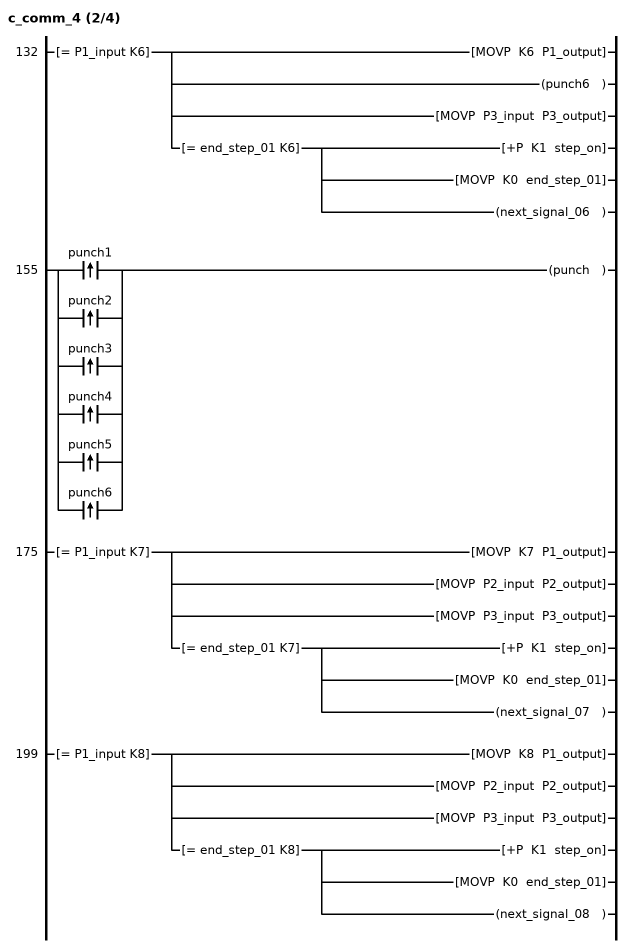
[picture p48: ladder of c_comm_4, rungs at steps 132 to 199]
132   LD=     P1_input K6
      MOVP    K6 P1_output
      OUT     punch6
      MOVP    P3_input P3_output
      AND=    end_step_01 K6
      +P      K1 step_on
      MOVP    K0 end_step_01
      OUT     next_signal_06
155   LDP     punch1
      ORP     punch2
      ORP     punch3
      ORP     punch4
      ORP     punch5
      ORP     punch6
      OUT     punch
175   LD=     P1_input K7
      MOVP    K7 P1_output
      MOVP    P2_input P2_output
      MOVP    P3_input P3_output
      AND=    end_step_01 K7
      +P      K1 step_on
      MOVP    K0 end_step_01
      OUT     next_signal_07
199   LD=     P1_input K8
      MOVP    K8 P1_output
      MOVP    P2_input P2_output
      MOVP    P3_input P3_output
      AND=    end_step_01 K8
      +P      K1 step_on
      MOVP    K0 end_step_01
      OUT     next_signal_08
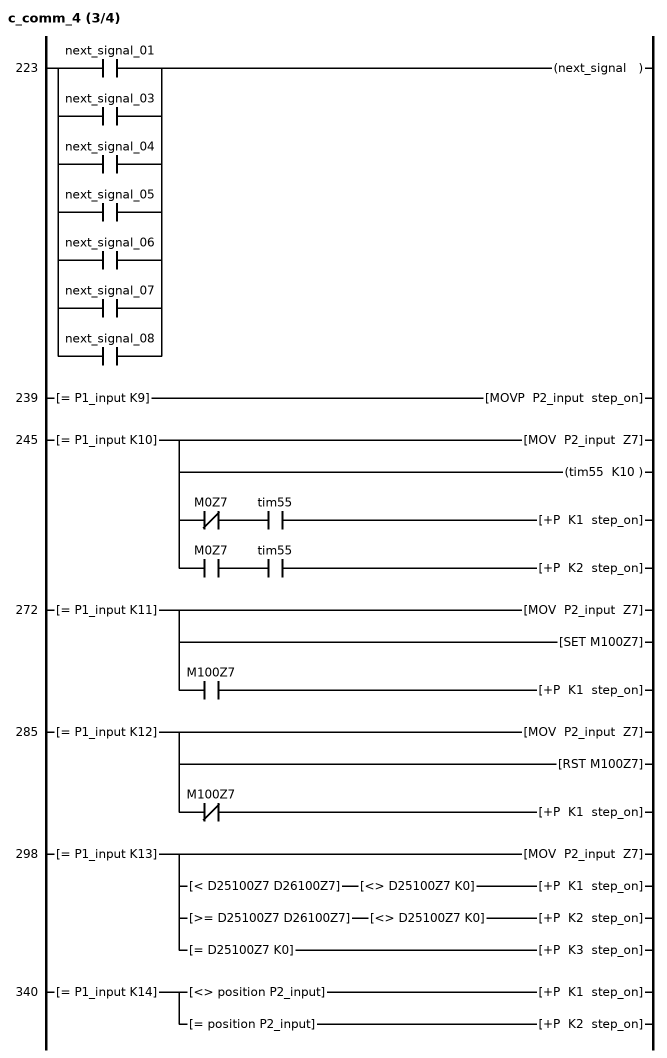
223   LD      next_signal_01
      OR      next_signal_03
      OR      next_signal_04
      OR      next_signal_05
      OR      next_signal_06
      OR      next_signal_07
      OR      next_signal_08
      OUT     next_signal
239   LD=     P1_input K9
      MOVP    P2_input step_on
245   LD=     P1_input K10
      MOV     P2_input Z7
      OUT     tim55 K10
      MPS
      ANI     M0Z7
      AND     tim55
      +P      K1 step_on
      MPP
      AND     M0Z7
      AND     tim55
      +P      K2 step_on
272   LD=     P1_input K11
      MOV     P2_input Z7
      SET     M100Z7
      AND     M100Z7
      +P      K1 step_on
285   LD=     P1_input K12
      MOV     P2_input Z7
      RST     M100Z7
      ANI     M100Z7
      +P      K1 step_on
298   LD=     P1_input K13
      MOV     P2_input Z7
      MPS
      AND<    D25100Z7 D26100Z7
      AND<>   D25100Z7 K0
      +P      K1 step_on
      MRD
      AND>=   D25100Z7 D26100Z7
      AND<>   D25100Z7 K0
      +P      K2 step_on
      MPP
      AND=    D25100Z7 K0
      +P      K3 step_on
340   LD=     P1_input K14
      MPS
      AND<>   position P2_input
      +P      K1 step_on
      MPP
      AND=    position P2_input
      +P      K2 step_on
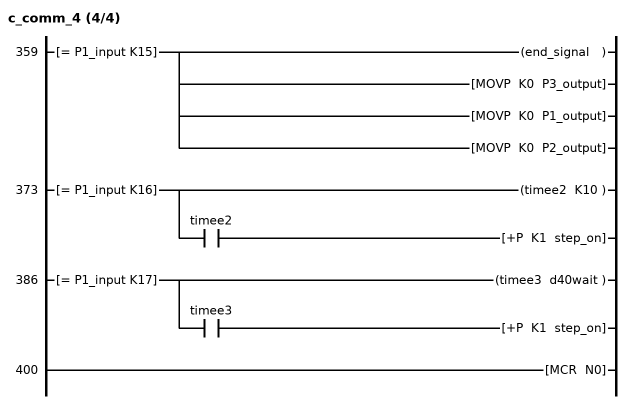
359   LD=     P1_input K15
      OUT     end_signal
      MOVP    K0 P3_output
      MOVP    K0 P1_output
      MOVP    K0 P2_output
373   LD=     P1_input K16
      OUT     timee2 K10
      AND     timee2
      +P      K1 step_on
386   LD=     P1_input K17
      OUT     timee3 d40wait
      AND     timee3
      +P      K1 step_on
400   MCR     N0
END_FUNCTION_BLOCK

PROGRAM carrier_1
VAR
  c_comm_1 : c_comm_1;
END_VAR
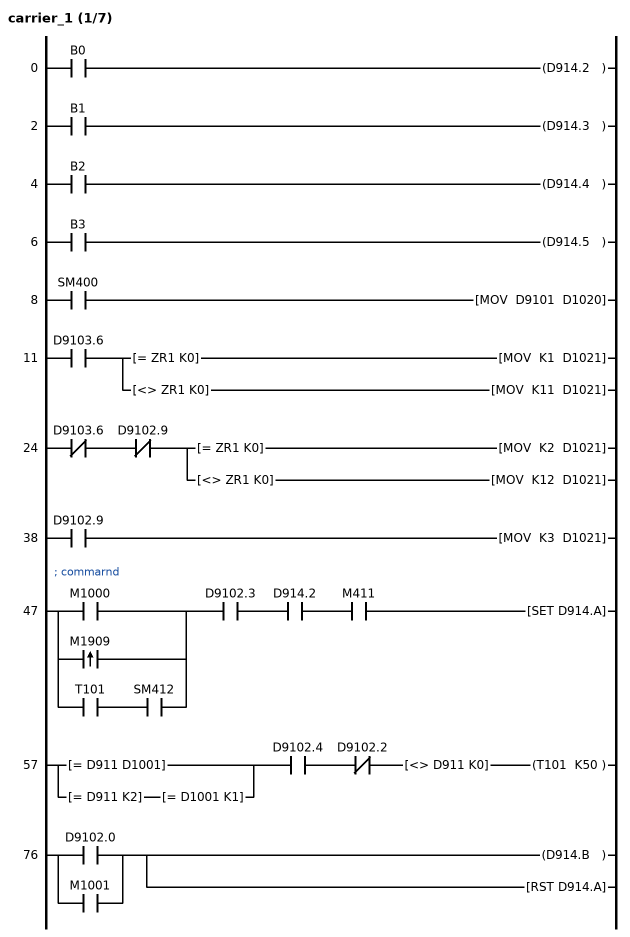
0     LD      B0
      OUT     D914.2
2     LD      B1
      OUT     D914.3
4     LD      B2
      OUT     D914.4
6     LD      B3
      OUT     D914.5
8     LD      SM400
      MOV     D9101 D1020
11    LD      D9103.6
      MPS
      AND=    ZR1 K0
      MOV     K1 D1021
      MPP
      AND<>   ZR1 K0
      MOV     K11 D1021
24    LDI     D9103.6
      ANI     D9102.9
      MPS
      AND=    ZR1 K0
      MOV     K2 D1021
      MPP
      AND<>   ZR1 K0
      MOV     K12 D1021
38    LD      D9102.9
      MOV     K3 D1021
; commarnd
47    LD      M1000
      ORP     M1909
      LD      T101
      AND     SM412
      ORB
      AND     D9102.3
      AND     D914.2
      AND     M411
      SET     D914.A
57    LD=     D911 D1001
      LD=     D911 K2
      AND=    D1001 K1
      ORB
      AND     D9102.4
      ANI     D9102.2
      AND<>   D911 K0
      OUT     T101 K50
76    LD      D9102.0
      OR      M1001
      OUT     D914.B
      RST     D914.A
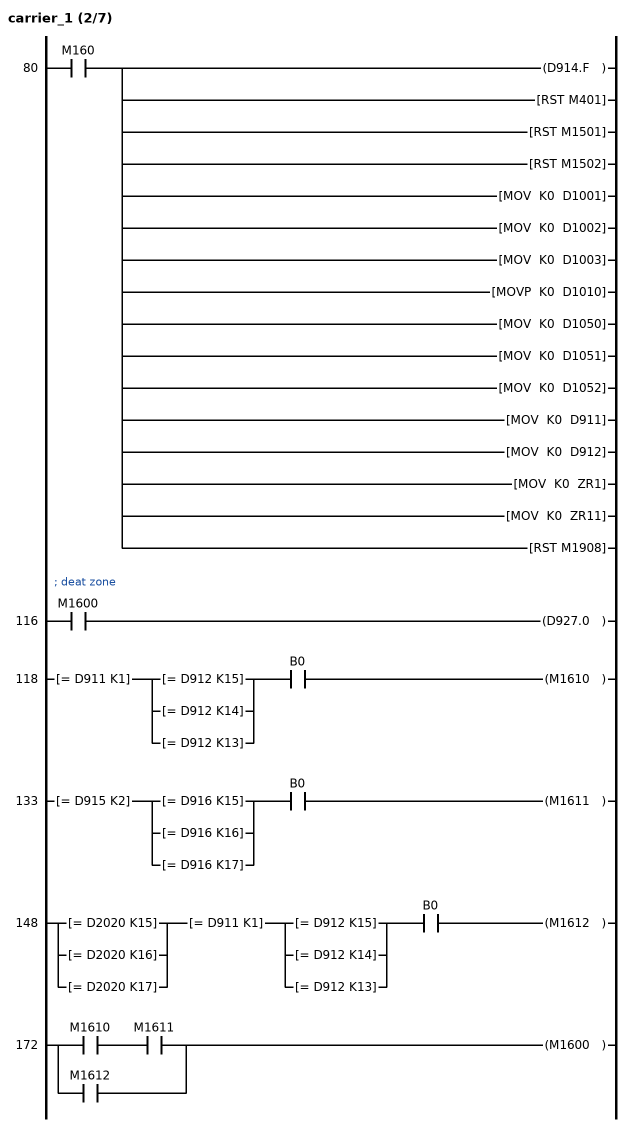
80    LD      M160
      OUT     D914.F
      RST     M401
      RST     M1501
      RST     M1502
      MOV     K0 D1001
      MOV     K0 D1002
      MOV     K0 D1003
      MOVP    K0 D1010
      MOV     K0 D1050
      MOV     K0 D1051
      MOV     K0 D1052
      MOV     K0 D911
      MOV     K0 D912
      MOV     K0 ZR1
      MOV     K0 ZR11
      RST     M1908
; deat zone
116   LD      M1600
      OUT     D927.0
118   LD=     D911 K1
      LD=     D912 K15
      OR=     D912 K14
      OR=     D912 K13
      ANB
      AND     B0
      OUT     M1610
133   LD=     D915 K2
      LD=     D916 K15
      OR=     D916 K16
      OR=     D916 K17
      ANB
      AND     B0
      OUT     M1611
148   LD=     D2020 K15
      OR=     D2020 K16
      OR=     D2020 K17
      AND=    D911 K1
      LD=     D912 K15
      OR=     D912 K14
      OR=     D912 K13
      ANB
      AND     B0
      OUT     M1612
172   LD      M1610
      AND     M1611
      OR      M1612
      OUT     M1600
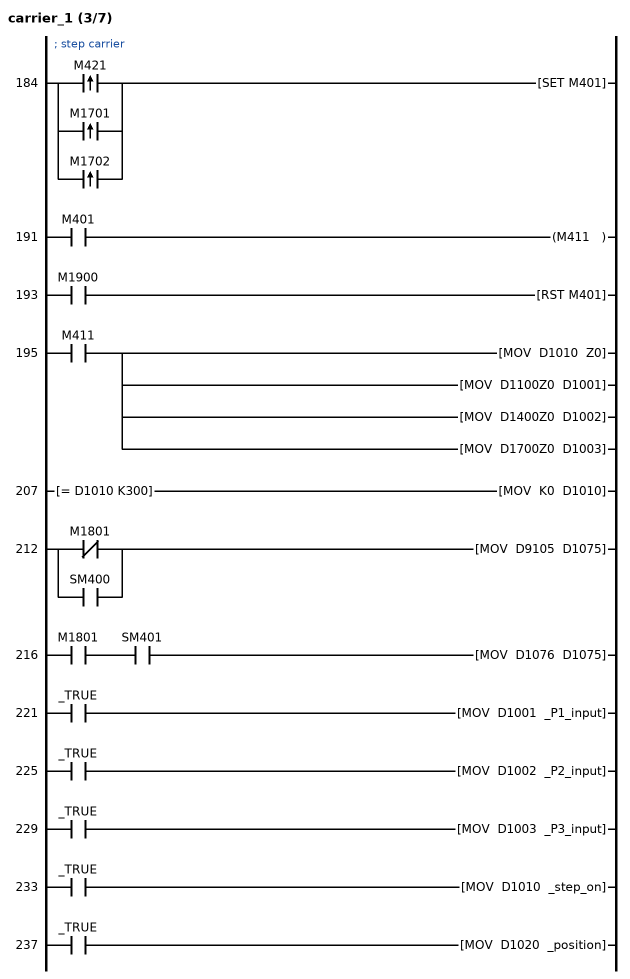
; step carrier
184   LDP     M421
      ORP     M1701
      ORP     M1702
      SET     M401
191   LD      M401
      OUT     M411
193   LD      M1900
      RST     M401
195   LD      M411
      MOV     D1010 Z0
      MOV     D1100Z0 D1001
      MOV     D1400Z0 D1002
      MOV     D1700Z0 D1003
207   LD=     D1010 K300
      MOV     K0 D1010
212   LDI     M1801
      OR      SM400
      MOV     D9105 D1075
216   LD      M1801
      AND     SM401
      MOV     D1076 D1075
; FB BLK START c_comm_1(c_comm_1)
221   LD      _TRUE
      MOV     D1001 _P1_input
225   LD      _TRUE
      MOV     D1002 _P2_input
229   LD      _TRUE
      MOV     D1003 _P3_input
233   LD      _TRUE
      MOV     D1010 _step_on
237   LD      _TRUE
      MOV     D1020 _position
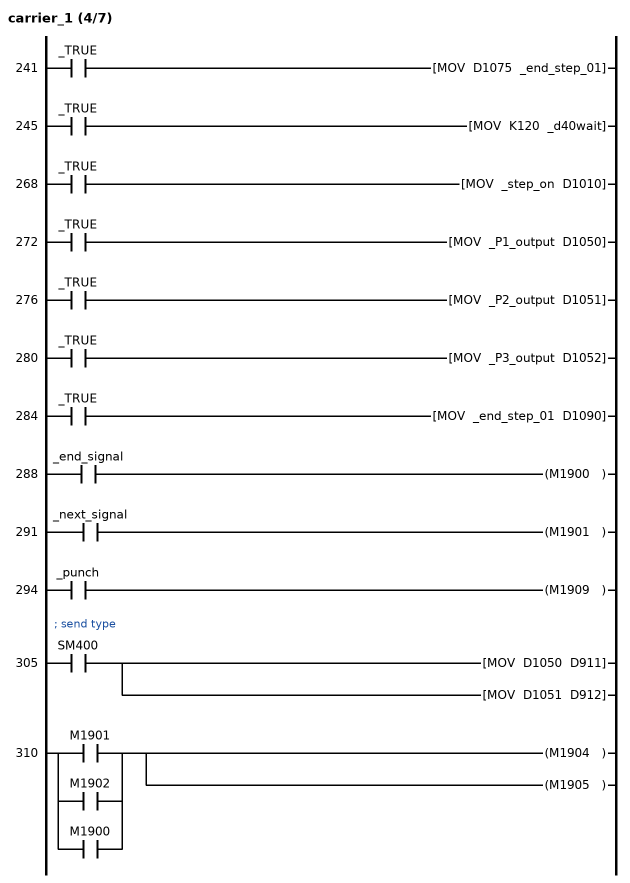
241   LD      _TRUE
      MOV     D1075 _end_step_01
245   LD      _TRUE
      MOV     K120 _d40wait
; FB START
; FB_NAME c_comm_1
; INSTANCE_NAME c_comm_1
; FB IN_W:P1_input
; FB OUT_step_on:W
; FB IN_W:P2_input
; FB OUT_P1_output:W
; FB IN_W:P3_input
; FB OUT_P2_output:W
; FB IN_W:step_on
; FB OUT_P3_output:W
; FB IN_W:position
; FB OUT_end_step_01:W
; FB IN_W:end_step_01
; FB OUT_end_signal:B
; FB IN_W:d40wait
; FB OUT_next_signal:B
; FB OUT_punch:B
; FB END
268   LD      _TRUE
      MOV     _step_on D1010
272   LD      _TRUE
      MOV     _P1_output D1050
276   LD      _TRUE
      MOV     _P2_output D1051
280   LD      _TRUE
      MOV     _P3_output D1052
284   LD      _TRUE
      MOV     _end_step_01 D1090
288   LD      _end_signal
      OUT     M1900
291   LD      _next_signal
      OUT     M1901
294   LD      _punch
      OUT     M1909
; FB BLK END
; send type
305   LD      SM400
      MOV     D1050 D911
      MOV     D1051 D912
310   LD      M1901
      OR      M1902
      OR      M1900
      OUT     M1904
      OUT     M1905
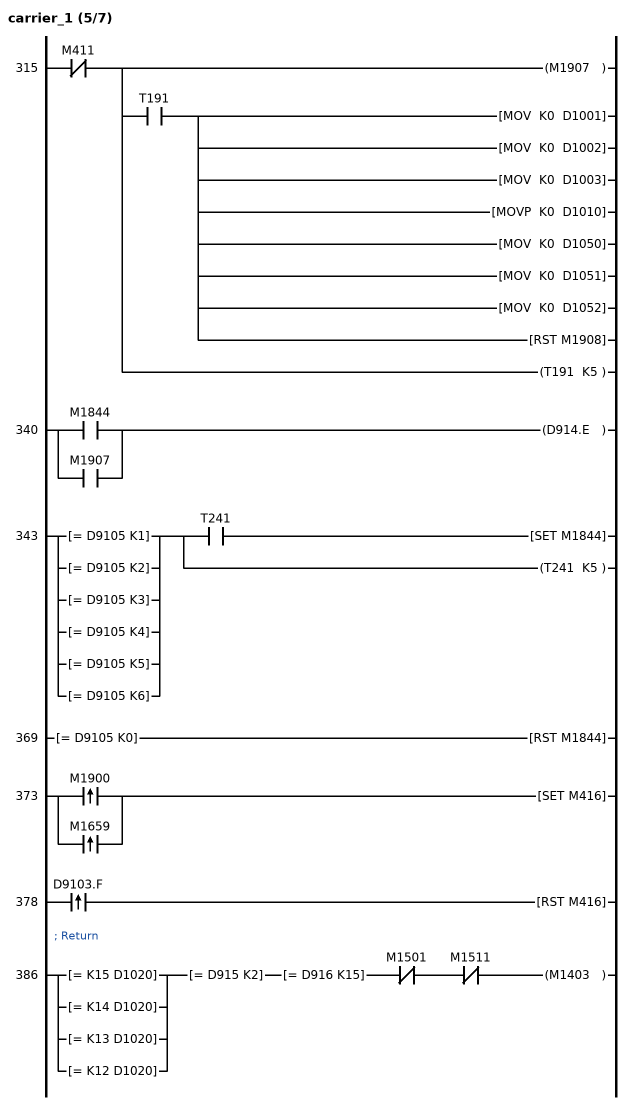
315   LDI     M411
      OUT     M1907
      MPS
      AND     T191
      MOV     K0 D1001
      MOV     K0 D1002
      MOV     K0 D1003
      MOVP    K0 D1010
      MOV     K0 D1050
      MOV     K0 D1051
      MOV     K0 D1052
      RST     M1908
      MPP
      OUT     T191 K5
340   LD      M1844
      OR      M1907
      OUT     D914.E
343   LD=     D9105 K1
      OR=     D9105 K2
      OR=     D9105 K3
      OR=     D9105 K4
      OR=     D9105 K5
      OR=     D9105 K6
      MPS
      AND     T241
      SET     M1844
      MPP
      OUT     T241 K5
369   LD=     D9105 K0
      RST     M1844
373   LDP     M1900
      ORP     M1659
      SET     M416
378   LDP     D9103.F
      RST     M416
; Return
386   LD=     K15 D1020
      OR=     K14 D1020
      OR=     K13 D1020
      OR=     K12 D1020
      AND=    D915 K2
      AND=    D916 K15
      ANI     M1501
      ANI     M1511
      OUT     M1403
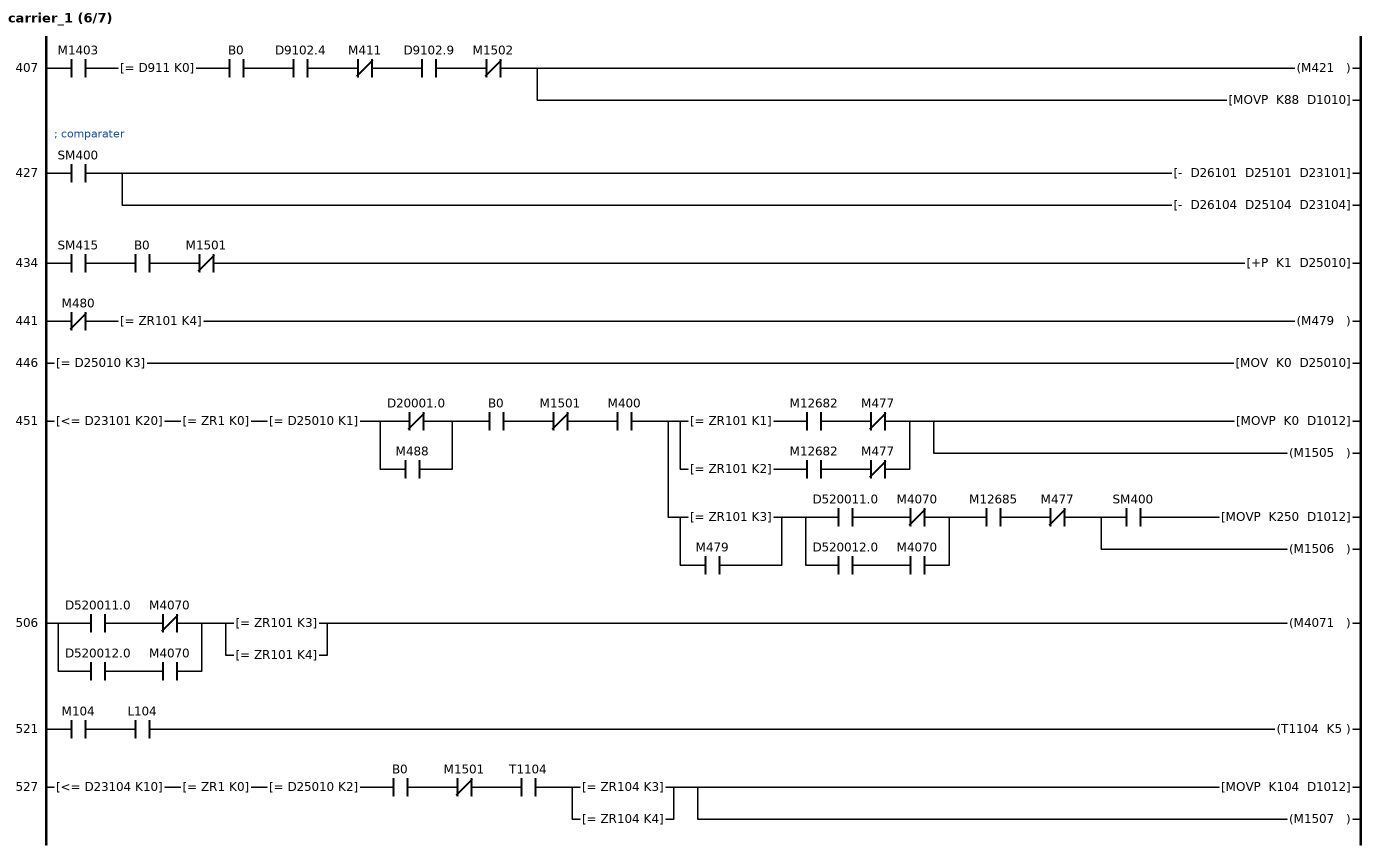
407   LD      M1403
      AND=    D911 K0
      AND     B0
      AND     D9102.4
      ANI     M411
      AND     D9102.9
      ANI     M1502
      OUT     M421
      MOVP    K88 D1010
; comparater
427   LD      SM400
      -       D26101 D25101 D23101
      -       D26104 D25104 D23104
434   LD      SM415
      AND     B0
      ANI     M1501
      +P      K1 D25010
441   LDI     M480
      AND=    ZR101 K4
      OUT     M479
446   LD=     D25010 K3
      MOV     K0 D25010
451   LD<=    D23101 K20
      AND=    ZR1 K0
      AND=    D25010 K1
      LDI     D20001.0
      OR      M488
      ANB
      AND     B0
      ANI     M1501
      AND     M400
      MPS
      LD=     ZR101 K1
      AND     M12682
      ANI     M477
      LD=     ZR101 K2
      AND     M12682
      ANI     M477
      ORB
      ANB
      MOVP    K0 D1012
      OUT     M1505
      MPP
      LD=     ZR101 K3
      OR      M479
      ANB
      LD      D520011.0
      ANI     M4070
      LD      D520012.0
      AND     M4070
      ORB
      ANB
      AND     M12685
      ANI     M477
      MPS
      AND     SM400
      MOVP    K250 D1012
      MPP
      OUT     M1506
506   LD      D520011.0
      ANI     M4070
      LD      D520012.0
      AND     M4070
      ORB
      LD=     ZR101 K3
      OR=     ZR101 K4
      ANB
      OUT     M4071
521   LD      M104
      AND     L104
      OUT     T1104 K5
527   LD<=    D23104 K10
      AND=    ZR1 K0
      AND=    D25010 K2
      AND     B0
      ANI     M1501
      AND     T1104
      LD=     ZR104 K3
      OR=     ZR104 K4
      ANB
      MOVP    K104 D1012
      OUT     M1507
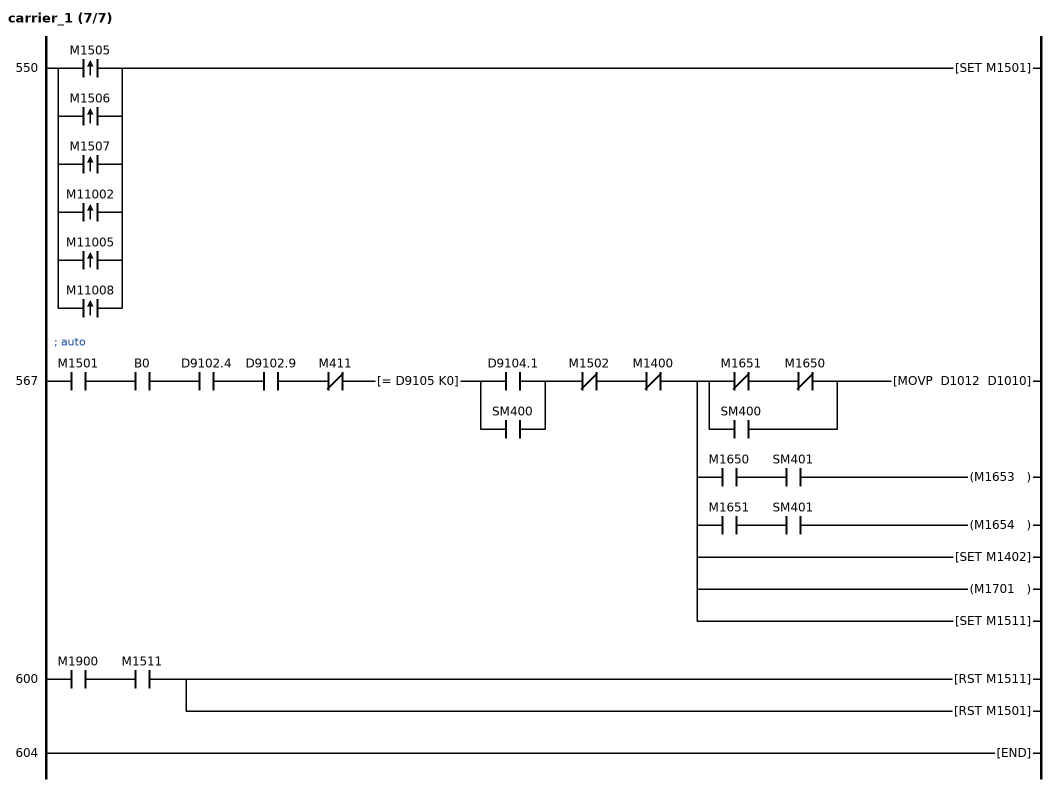
550   LDP     M1505
      ORP     M1506
      ORP     M1507
      ORP     M11002
      ORP     M11005
      ORP     M11008
      SET     M1501
; auto
567   LD      M1501
      AND     B0
      AND     D9102.4
      AND     D9102.9
      ANI     M411
      AND=    D9105 K0
      LD      D9104.1
      OR      SM400
      ANB
      ANI     M1502
      ANI     M1400
      MPS
      LDI     M1651
      ANI     M1650
      OR      SM400
      ANB
      MOVP    D1012 D1010
      MRD
      AND     M1650
      AND     SM401
      OUT     M1653
      MRD
      AND     M1651
      AND     SM401
      OUT     M1654
      MPP
      SET     M1402
      OUT     M1701
      SET     M1511
600   LD      M1900
      AND     M1511
      RST     M1511
      RST     M1501
604   END
END_PROGRAM

PROGRAM carrier_2
VAR
  c_comm_2 : c_comm_2;
END_VAR
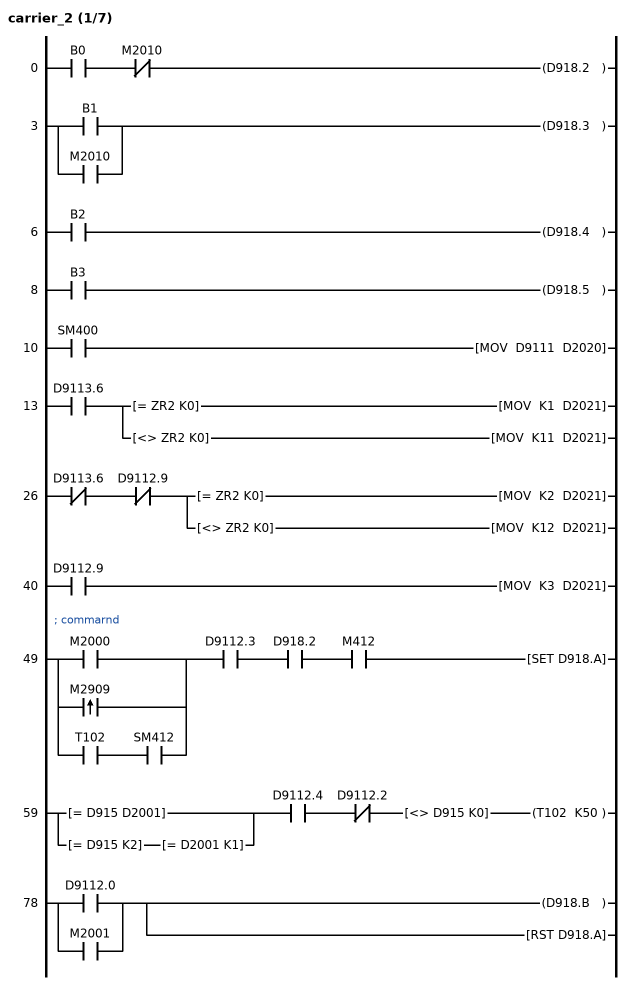
0     LD      B0
      ANI     M2010
      OUT     D918.2
3     LD      B1
      OR      M2010
      OUT     D918.3
6     LD      B2
      OUT     D918.4
8     LD      B3
      OUT     D918.5
10    LD      SM400
      MOV     D9111 D2020
13    LD      D9113.6
      MPS
      AND=    ZR2 K0
      MOV     K1 D2021
      MPP
      AND<>   ZR2 K0
      MOV     K11 D2021
26    LDI     D9113.6
      ANI     D9112.9
      MPS
      AND=    ZR2 K0
      MOV     K2 D2021
      MPP
      AND<>   ZR2 K0
      MOV     K12 D2021
40    LD      D9112.9
      MOV     K3 D2021
; commarnd
49    LD      M2000
      ORP     M2909
      LD      T102
      AND     SM412
      ORB
      AND     D9112.3
      AND     D918.2
      AND     M412
      SET     D918.A
59    LD=     D915 D2001
      LD=     D915 K2
      AND=    D2001 K1
      ORB
      AND     D9112.4
      ANI     D9112.2
      AND<>   D915 K0
      OUT     T102 K50
78    LD      D9112.0
      OR      M2001
      OUT     D918.B
      RST     D918.A
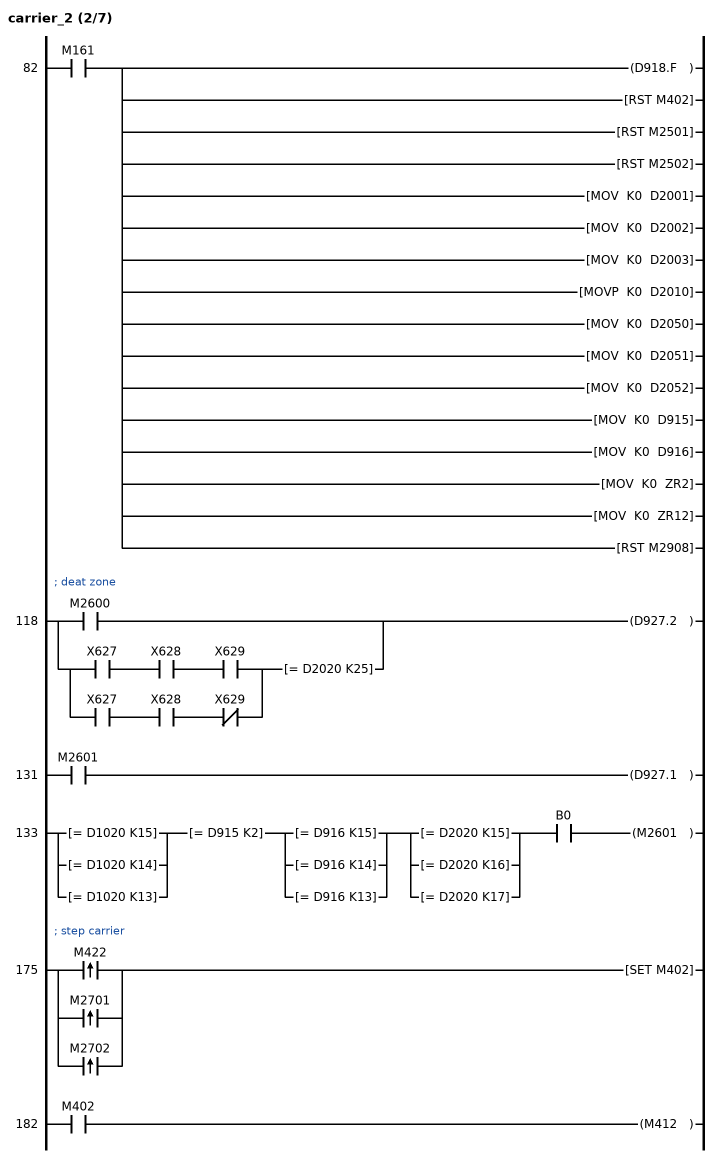
82    LD      M161
      OUT     D918.F
      RST     M402
      RST     M2501
      RST     M2502
      MOV     K0 D2001
      MOV     K0 D2002
      MOV     K0 D2003
      MOVP    K0 D2010
      MOV     K0 D2050
      MOV     K0 D2051
      MOV     K0 D2052
      MOV     K0 D915
      MOV     K0 D916
      MOV     K0 ZR2
      MOV     K0 ZR12
      RST     M2908
; deat zone
118   LD      M2600
      LD      X627
      AND     X628
      AND     X629
      LD      X627
      AND     X628
      ANI     X629
      ORB
      AND=    D2020 K25
      ORB
      OUT     D927.2
131   LD      M2601
      OUT     D927.1
133   LD=     D1020 K15
      OR=     D1020 K14
      OR=     D1020 K13
      AND=    D915 K2
      LD=     D916 K15
      OR=     D916 K14
      OR=     D916 K13
      ANB
      LD=     D2020 K15
      OR=     D2020 K16
      OR=     D2020 K17
      ANB
      AND     B0
      OUT     M2601
; step carrier
175   LDP     M422
      ORP     M2701
      ORP     M2702
      SET     M402
182   LD      M402
      OUT     M412
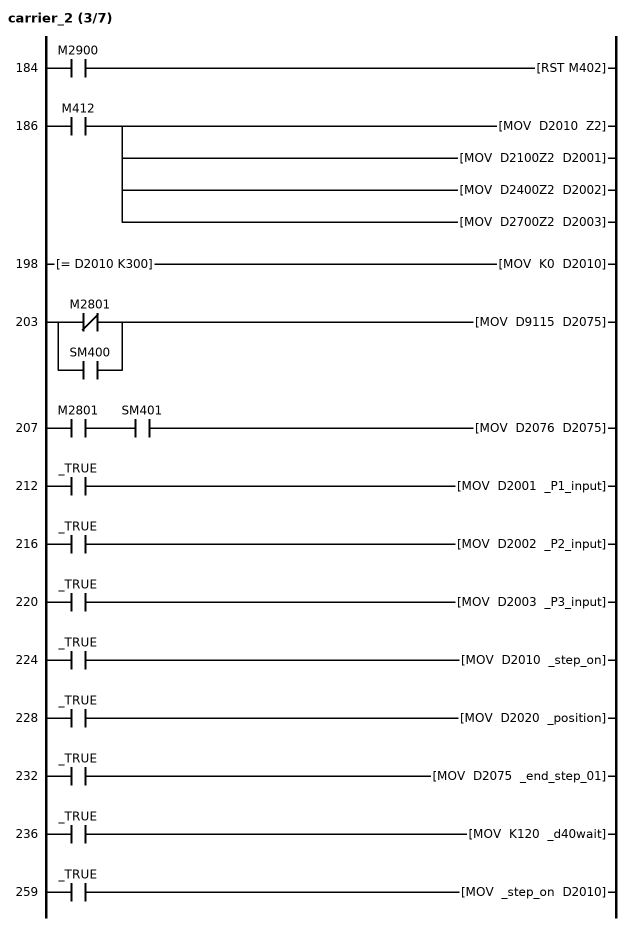
184   LD      M2900
      RST     M402
186   LD      M412
      MOV     D2010 Z2
      MOV     D2100Z2 D2001
      MOV     D2400Z2 D2002
      MOV     D2700Z2 D2003
198   LD=     D2010 K300
      MOV     K0 D2010
203   LDI     M2801
      OR      SM400
      MOV     D9115 D2075
207   LD      M2801
      AND     SM401
      MOV     D2076 D2075
; FB BLK START c_comm_2(c_comm_2)
212   LD      _TRUE
      MOV     D2001 _P1_input
216   LD      _TRUE
      MOV     D2002 _P2_input
220   LD      _TRUE
      MOV     D2003 _P3_input
224   LD      _TRUE
      MOV     D2010 _step_on
228   LD      _TRUE
      MOV     D2020 _position
232   LD      _TRUE
      MOV     D2075 _end_step_01
236   LD      _TRUE
      MOV     K120 _d40wait
; FB START
; FB_NAME c_comm_2
; INSTANCE_NAME c_comm_2
; FB IN_W:P1_input
; FB OUT_step_on:W
; FB IN_W:P2_input
; FB OUT_P1_output:W
; FB IN_W:P3_input
; FB OUT_P2_output:W
; FB IN_W:step_on
; FB OUT_P3_output:W
; FB IN_W:position
; FB OUT_end_step_01:W
; FB IN_W:end_step_01
; FB OUT_end_signal:B
; FB IN_W:d40wait
; FB OUT_next_signal:B
; FB OUT_punch:B
; FB END
259   LD      _TRUE
      MOV     _step_on D2010
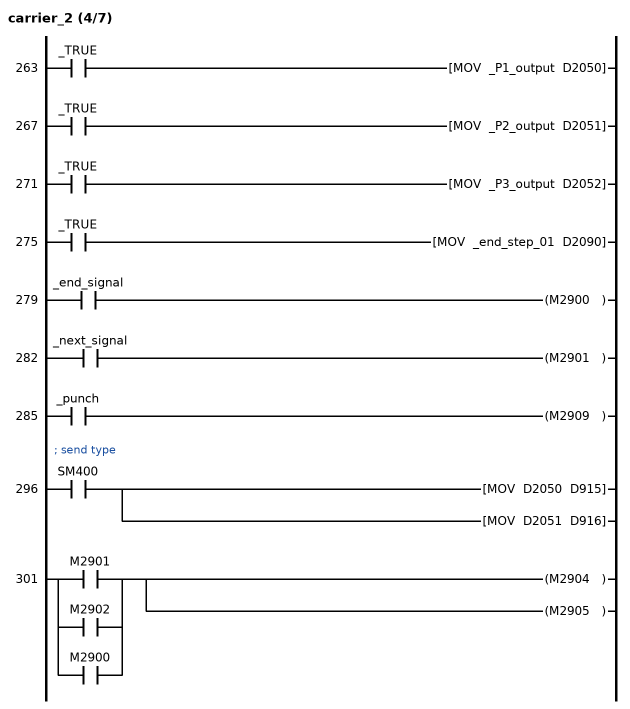
263   LD      _TRUE
      MOV     _P1_output D2050
267   LD      _TRUE
      MOV     _P2_output D2051
271   LD      _TRUE
      MOV     _P3_output D2052
275   LD      _TRUE
      MOV     _end_step_01 D2090
279   LD      _end_signal
      OUT     M2900
282   LD      _next_signal
      OUT     M2901
285   LD      _punch
      OUT     M2909
; FB BLK END
; send type
296   LD      SM400
      MOV     D2050 D915
      MOV     D2051 D916
301   LD      M2901
      OR      M2902
      OR      M2900
      OUT     M2904
      OUT     M2905
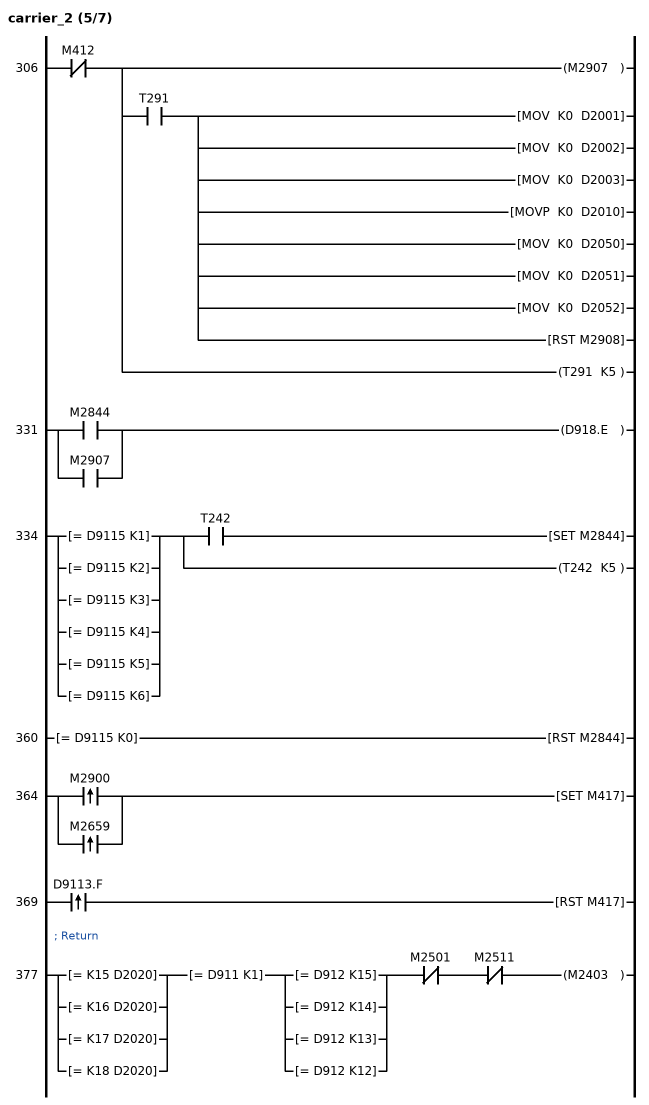
306   LDI     M412
      OUT     M2907
      MPS
      AND     T291
      MOV     K0 D2001
      MOV     K0 D2002
      MOV     K0 D2003
      MOVP    K0 D2010
      MOV     K0 D2050
      MOV     K0 D2051
      MOV     K0 D2052
      RST     M2908
      MPP
      OUT     T291 K5
331   LD      M2844
      OR      M2907
      OUT     D918.E
334   LD=     D9115 K1
      OR=     D9115 K2
      OR=     D9115 K3
      OR=     D9115 K4
      OR=     D9115 K5
      OR=     D9115 K6
      MPS
      AND     T242
      SET     M2844
      MPP
      OUT     T242 K5
360   LD=     D9115 K0
      RST     M2844
364   LDP     M2900
      ORP     M2659
      SET     M417
369   LDP     D9113.F
      RST     M417
; Return
377   LD=     K15 D2020
      OR=     K16 D2020
      OR=     K17 D2020
      OR=     K18 D2020
      AND=    D911 K1
      LD=     D912 K15
      OR=     D912 K14
      OR=     D912 K13
      OR=     D912 K12
      ANB
      ANI     M2501
      ANI     M2511
      OUT     M2403
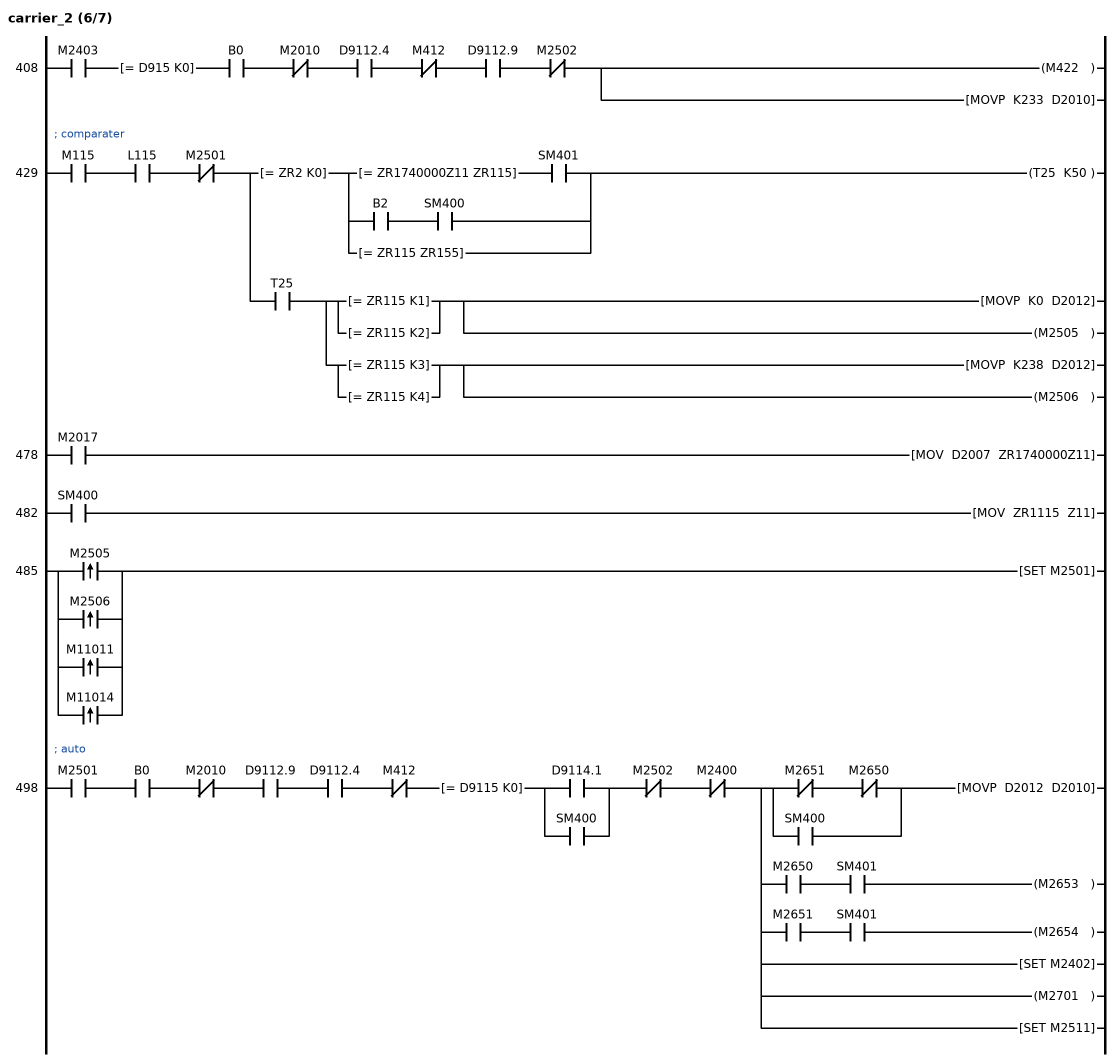
408   LD      M2403
      AND=    D915 K0
      AND     B0
      ANI     M2010
      AND     D9112.4
      ANI     M412
      AND     D9112.9
      ANI     M2502
      OUT     M422
      MOVP    K233 D2010
; comparater
429   LD      M115
      AND     L115
      ANI     M2501
      MPS
      AND=    ZR2 K0
      LD=     ZR1740000Z11 ZR115
      AND     SM401
      LD      B2
      AND     SM400
      ORB
      OR=     ZR115 ZR155
      ANB
      OUT     T25 K50
      MPP
      AND     T25
      MPS
      LD=     ZR115 K1
      OR=     ZR115 K2
      ANB
      MOVP    K0 D2012
      OUT     M2505
      MPP
      LD=     ZR115 K3
      OR=     ZR115 K4
      ANB
      MOVP    K238 D2012
      OUT     M2506
478   LD      M2017
      MOV     D2007 ZR1740000Z11
482   LD      SM400
      MOV     ZR1115 Z11
485   LDP     M2505
      ORP     M2506
      ORP     M11011
      ORP     M11014
      SET     M2501
; auto
498   LD      M2501
      AND     B0
      ANI     M2010
      AND     D9112.9
      AND     D9112.4
      ANI     M412
      AND=    D9115 K0
      LD      D9114.1
      OR      SM400
      ANB
      ANI     M2502
      ANI     M2400
      MPS
      LDI     M2651
      ANI     M2650
      OR      SM400
      ANB
      MOVP    D2012 D2010
      MRD
      AND     M2650
      AND     SM401
      OUT     M2653
      MRD
      AND     M2651
      AND     SM401
      OUT     M2654
      MPP
      SET     M2402
      OUT     M2701
      SET     M2511
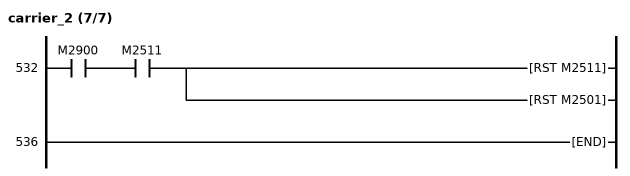
532   LD      M2900
      AND     M2511
      RST     M2511
      RST     M2501
536   END
END_PROGRAM

PROGRAM carrier_3
VAR
  c_comm_3 : c_comm_3;
  __IST_76367eaf8b844e8d : I+ST_76367eaf8b844e8d;
  __IST_4f96081e274e4d1c : I+ST_4f96081e274e4d1c;
END_VAR
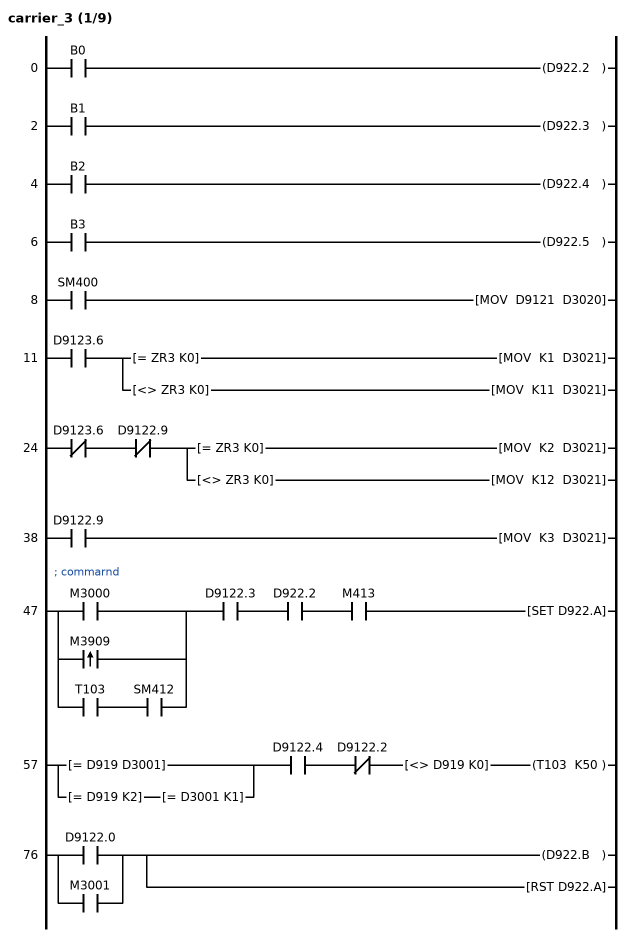
0     LD      B0
      OUT     D922.2
2     LD      B1
      OUT     D922.3
4     LD      B2
      OUT     D922.4
6     LD      B3
      OUT     D922.5
8     LD      SM400
      MOV     D9121 D3020
11    LD      D9123.6
      MPS
      AND=    ZR3 K0
      MOV     K1 D3021
      MPP
      AND<>   ZR3 K0
      MOV     K11 D3021
24    LDI     D9123.6
      ANI     D9122.9
      MPS
      AND=    ZR3 K0
      MOV     K2 D3021
      MPP
      AND<>   ZR3 K0
      MOV     K12 D3021
38    LD      D9122.9
      MOV     K3 D3021
; commarnd
47    LD      M3000
      ORP     M3909
      LD      T103
      AND     SM412
      ORB
      AND     D9122.3
      AND     D922.2
      AND     M413
      SET     D922.A
57    LD=     D919 D3001
      LD=     D919 K2
      AND=    D3001 K1
      ORB
      AND     D9122.4
      ANI     D9122.2
      AND<>   D919 K0
      OUT     T103 K50
76    LD      D9122.0
      OR      M3001
      OUT     D922.B
      RST     D922.A
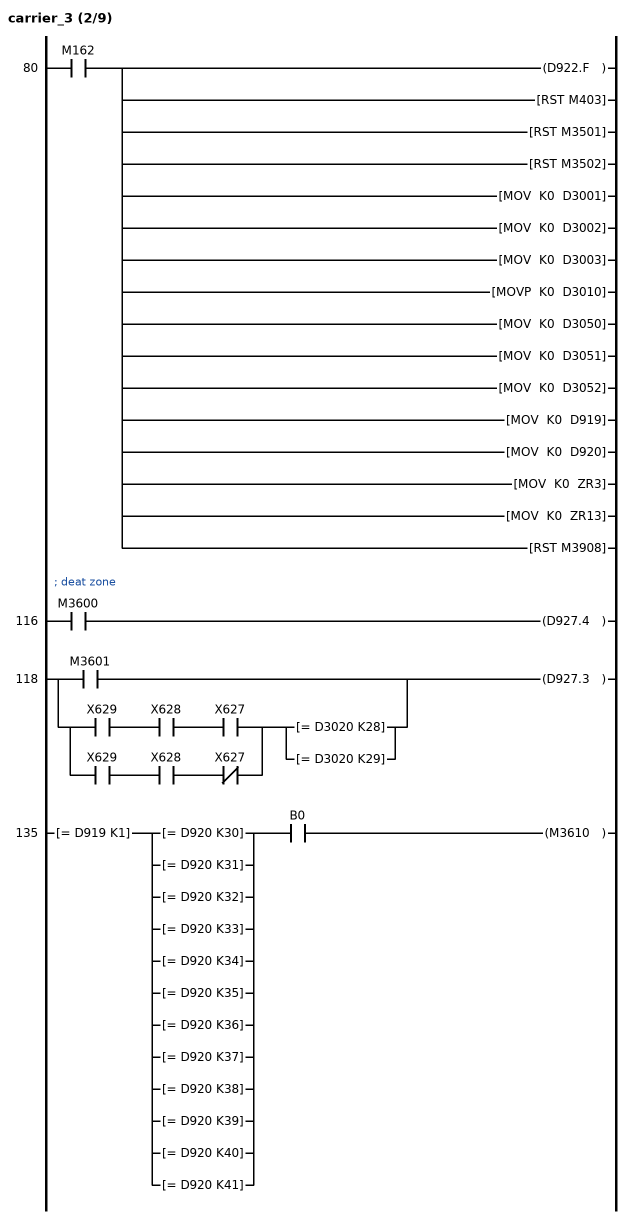
80    LD      M162
      OUT     D922.F
      RST     M403
      RST     M3501
      RST     M3502
      MOV     K0 D3001
      MOV     K0 D3002
      MOV     K0 D3003
      MOVP    K0 D3010
      MOV     K0 D3050
      MOV     K0 D3051
      MOV     K0 D3052
      MOV     K0 D919
      MOV     K0 D920
      MOV     K0 ZR3
      MOV     K0 ZR13
      RST     M3908
; deat zone
116   LD      M3600
      OUT     D927.4
118   LD      M3601
      LD      X629
      AND     X628
      AND     X627
      LD      X629
      AND     X628
      ANI     X627
      ORB
      LD=     D3020 K28
      OR=     D3020 K29
      ANB
      ORB
      OUT     D927.3
135   LD=     D919 K1
      LD=     D920 K30
      OR=     D920 K31
      OR=     D920 K32
      OR=     D920 K33
      OR=     D920 K34
      OR=     D920 K35
      OR=     D920 K36
      OR=     D920 K37
      OR=     D920 K38
      OR=     D920 K39
      OR=     D920 K40
      OR=     D920 K41
      ANB
      AND     B0
      OUT     M3610
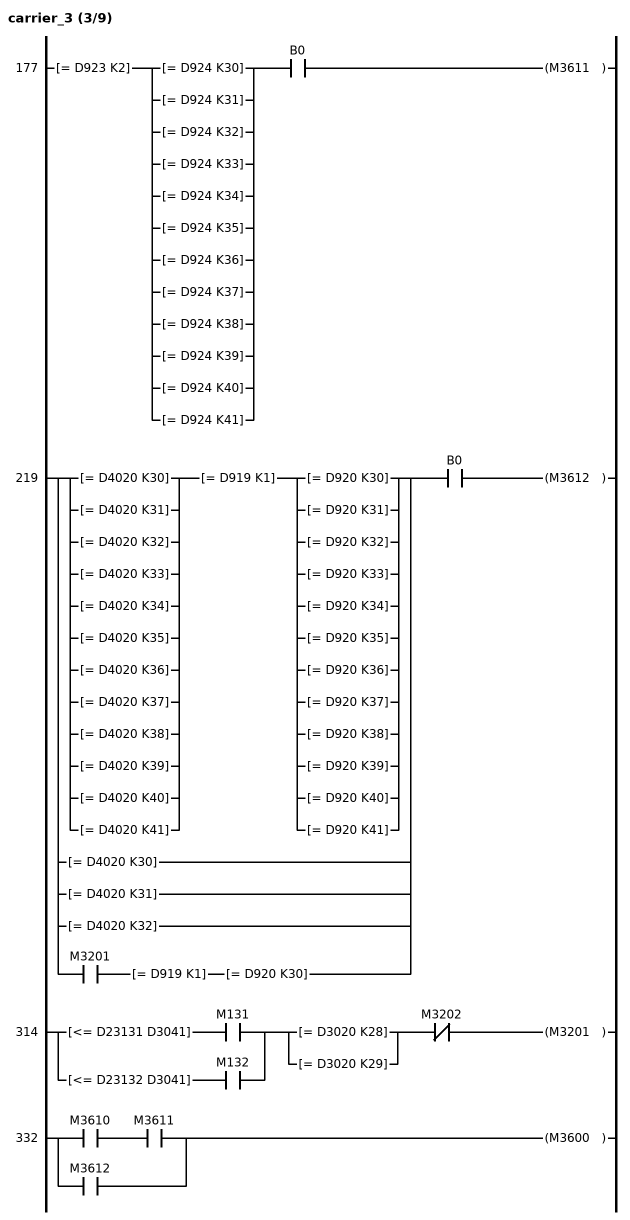
177   LD=     D923 K2
      LD=     D924 K30
      OR=     D924 K31
      OR=     D924 K32
      OR=     D924 K33
      OR=     D924 K34
      OR=     D924 K35
      OR=     D924 K36
      OR=     D924 K37
      OR=     D924 K38
      OR=     D924 K39
      OR=     D924 K40
      OR=     D924 K41
      ANB
      AND     B0
      OUT     M3611
219   LD=     D4020 K30
      OR=     D4020 K31
      OR=     D4020 K32
      OR=     D4020 K33
      OR=     D4020 K34
      OR=     D4020 K35
      OR=     D4020 K36
      OR=     D4020 K37
      OR=     D4020 K38
      OR=     D4020 K39
      OR=     D4020 K40
      OR=     D4020 K41
      AND=    D919 K1
      LD=     D920 K30
      OR=     D920 K31
      OR=     D920 K32
      OR=     D920 K33
      OR=     D920 K34
      OR=     D920 K35
      OR=     D920 K36
      OR=     D920 K37
      OR=     D920 K38
      OR=     D920 K39
      OR=     D920 K40
      OR=     D920 K41
      ANB
      OR=     D4020 K30
      OR=     D4020 K31
      OR=     D4020 K32
      LD      M3201
      AND=    D919 K1
      AND=    D920 K30
      ORB
      AND     B0
      OUT     M3612
314   LD<=    D23131 D3041
      AND     M131
      LD<=    D23132 D3041
      AND     M132
      ORB
      LD=     D3020 K28
      OR=     D3020 K29
      ANB
      ANI     M3202
      OUT     M3201
332   LD      M3610
      AND     M3611
      OR      M3612
      OUT     M3600
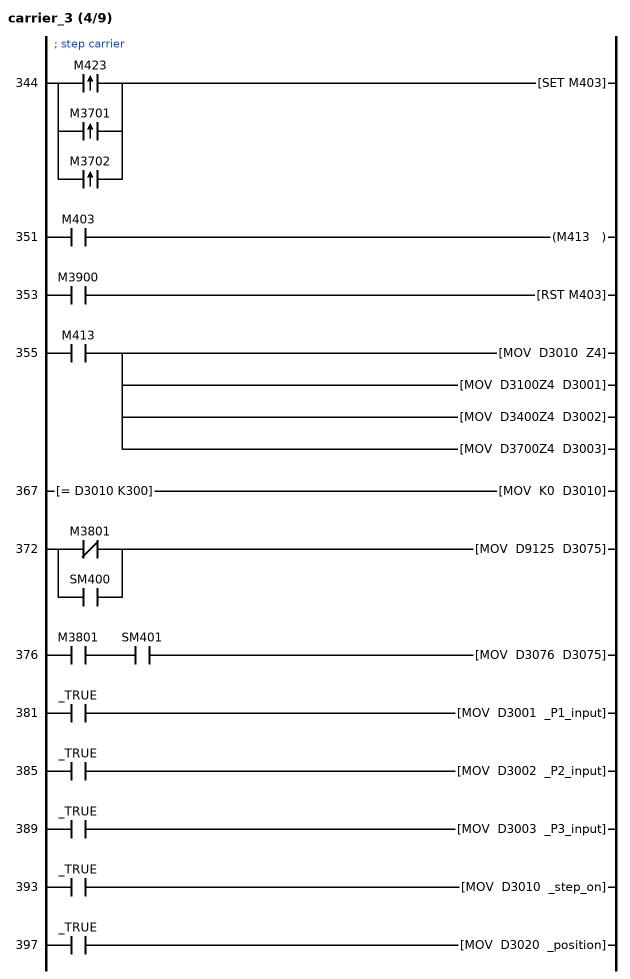
; step carrier
344   LDP     M423
      ORP     M3701
      ORP     M3702
      SET     M403
351   LD      M403
      OUT     M413
353   LD      M3900
      RST     M403
355   LD      M413
      MOV     D3010 Z4
      MOV     D3100Z4 D3001
      MOV     D3400Z4 D3002
      MOV     D3700Z4 D3003
367   LD=     D3010 K300
      MOV     K0 D3010
372   LDI     M3801
      OR      SM400
      MOV     D9125 D3075
376   LD      M3801
      AND     SM401
      MOV     D3076 D3075
; FB BLK START c_comm_3(c_comm_3)
381   LD      _TRUE
      MOV     D3001 _P1_input
385   LD      _TRUE
      MOV     D3002 _P2_input
389   LD      _TRUE
      MOV     D3003 _P3_input
393   LD      _TRUE
      MOV     D3010 _step_on
397   LD      _TRUE
      MOV     D3020 _position
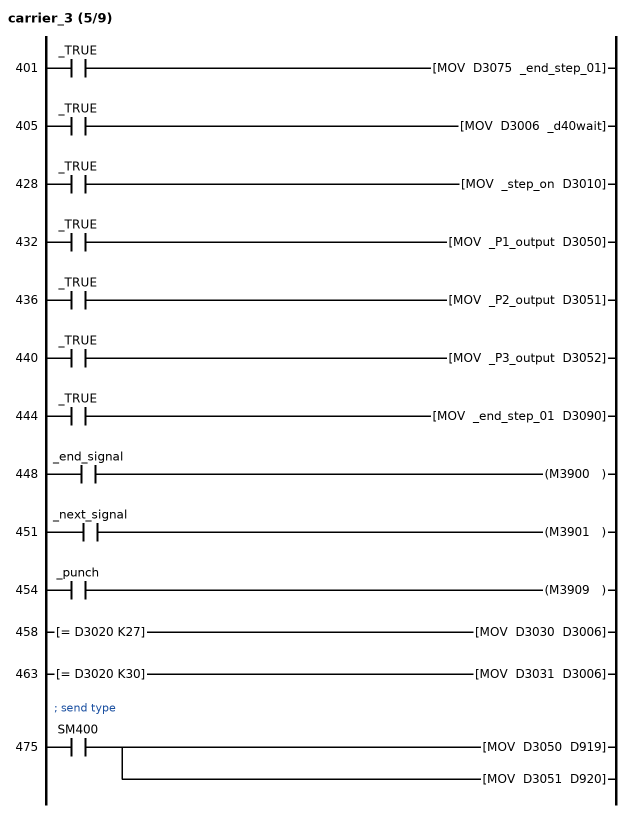
401   LD      _TRUE
      MOV     D3075 _end_step_01
405   LD      _TRUE
      MOV     D3006 _d40wait
; FB START
; FB_NAME c_comm_3
; INSTANCE_NAME c_comm_3
; FB IN_W:P1_input
; FB OUT_step_on:W
; FB IN_W:P2_input
; FB OUT_P1_output:W
; FB IN_W:P3_input
; FB OUT_P2_output:W
; FB IN_W:step_on
; FB OUT_P3_output:W
; FB IN_W:position
; FB OUT_end_step_01:W
; FB IN_W:end_step_01
; FB OUT_end_signal:B
; FB IN_W:d40wait
; FB OUT_next_signal:B
; FB OUT_punch:B
; FB END
428   LD      _TRUE
      MOV     _step_on D3010
432   LD      _TRUE
      MOV     _P1_output D3050
436   LD      _TRUE
      MOV     _P2_output D3051
440   LD      _TRUE
      MOV     _P3_output D3052
444   LD      _TRUE
      MOV     _end_step_01 D3090
448   LD      _end_signal
      OUT     M3900
451   LD      _next_signal
      OUT     M3901
454   LD      _punch
      OUT     M3909
; FB BLK END
458   LD=     D3020 K27
      MOV     D3030 D3006
463   LD=     D3020 K30
      MOV     D3031 D3006
; send type
475   LD      SM400
      MOV     D3050 D919
      MOV     D3051 D920
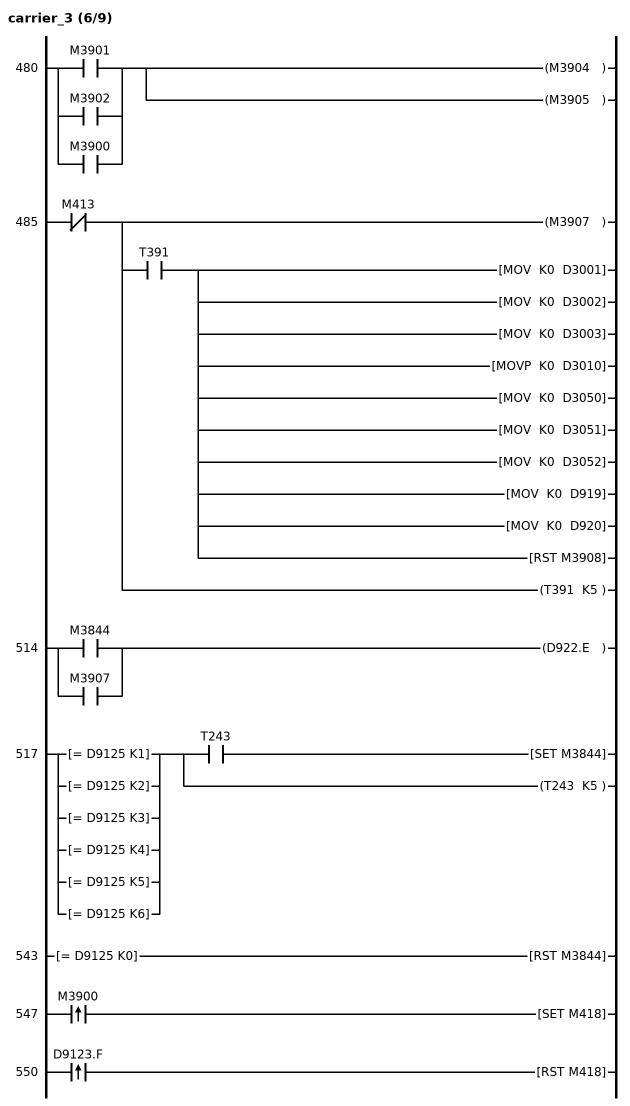
480   LD      M3901
      OR      M3902
      OR      M3900
      OUT     M3904
      OUT     M3905
485   LDI     M413
      OUT     M3907
      MPS
      AND     T391
      MOV     K0 D3001
      MOV     K0 D3002
      MOV     K0 D3003
      MOVP    K0 D3010
      MOV     K0 D3050
      MOV     K0 D3051
      MOV     K0 D3052
      MOV     K0 D919
      MOV     K0 D920
      RST     M3908
      MPP
      OUT     T391 K5
514   LD      M3844
      OR      M3907
      OUT     D922.E
517   LD=     D9125 K1
      OR=     D9125 K2
      OR=     D9125 K3
      OR=     D9125 K4
      OR=     D9125 K5
      OR=     D9125 K6
      MPS
      AND     T243
      SET     M3844
      MPP
      OUT     T243 K5
543   LD=     D9125 K0
      RST     M3844
547   LDP     M3900
      SET     M418
550   LDP     D9123.F
      RST     M418
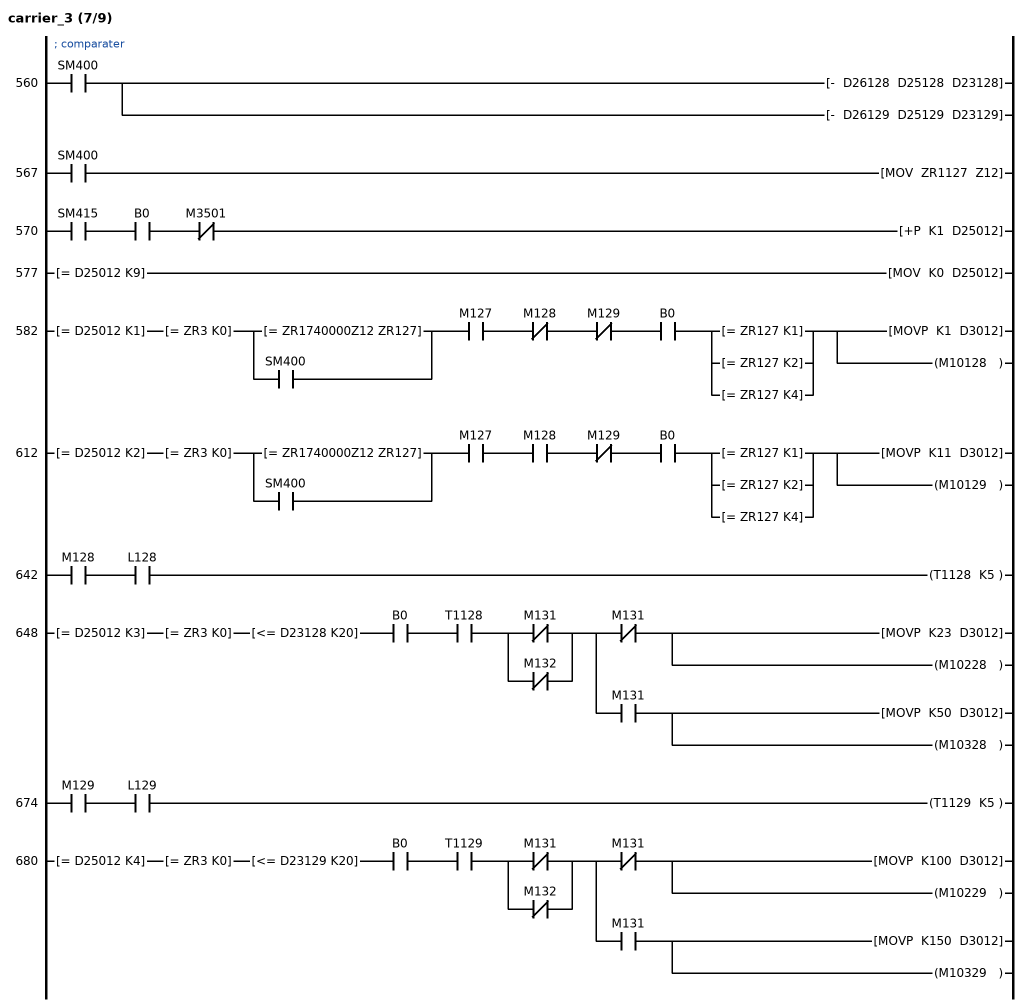
; comparater
560   LD      SM400
      -       D26128 D25128 D23128
      -       D26129 D25129 D23129
567   LD      SM400
      MOV     ZR1127 Z12
570   LD      SM415
      AND     B0
      ANI     M3501
      +P      K1 D25012
577   LD=     D25012 K9
      MOV     K0 D25012
582   LD=     D25012 K1
      AND=    ZR3 K0
      LD=     ZR1740000Z12 ZR127
      OR      SM400
      ANB
      AND     M127
      ANI     M128
      ANI     M129
      AND     B0
      LD=     ZR127 K1
      OR=     ZR127 K2
      OR=     ZR127 K4
      ANB
      MOVP    K1 D3012
      OUT     M10128
612   LD=     D25012 K2
      AND=    ZR3 K0
      LD=     ZR1740000Z12 ZR127
      OR      SM400
      ANB
      AND     M127
      AND     M128
      ANI     M129
      AND     B0
      LD=     ZR127 K1
      OR=     ZR127 K2
      OR=     ZR127 K4
      ANB
      MOVP    K11 D3012
      OUT     M10129
642   LD      M128
      AND     L128
      OUT     T1128 K5
648   LD=     D25012 K3
      AND=    ZR3 K0
      AND<=   D23128 K20
      AND     B0
      AND     T1128
      LDI     M131
      ORI     M132
      ANB
      MPS
      ANI     M131
      MOVP    K23 D3012
      OUT     M10228
      MPP
      AND     M131
      MOVP    K50 D3012
      OUT     M10328
674   LD      M129
      AND     L129
      OUT     T1129 K5
680   LD=     D25012 K4
      AND=    ZR3 K0
      AND<=   D23129 K20
      AND     B0
      AND     T1129
      LDI     M131
      ORI     M132
      ANB
      MPS
      ANI     M131
      MOVP    K100 D3012
      OUT     M10229
      MPP
      AND     M131
      MOVP    K150 D3012
      OUT     M10329
